// TIA Portal V16 export
// export: Created 2021-11-12T13:33:07.5254994Z, ExportSetting WithDefaults, DisplayName Totally Integrated Automation Portal, DisplayVersion V16 Update 3, DisplayName TIA Portal Version Control Interface, DisplayVersion V16 Update 2, DisplayName TIA Portal Openness, DisplayVersion V16 Update 3, DisplayName SINAMICS Startdrive Advanced, DisplayVersion V16 Update 5, DisplayName SINAMICS Startdrive G130, G150, S120, S150, SINAMICS MV, S210, DisplayVersion V16 Update 5, DisplayName SINAMICS Startdrive G110M, G120, G120C, G120D, G120P, G115D, DisplayVersion V16 Update 5, DisplayName STEP 7 Professional, DisplayVersion V16 Update 3, DisplayName STEP 7 Safety, DisplayVersion V16, DisplayName WinCC UA Professional, DisplayVersion V16 Update 3
DATA_BLOCK "HMI_PARAM_410"   // DB107
{ S7_Optimized_Access := 'TRUE' }
VERSION : 0.1
// stored: AutoNumber true, DBAccessibleFromOPCUA true, IsOnlyStoredInLoadMemory false, IsRetainMemResEnabled false, IsWriteProtectedInAS false, MemoryReserve 100
   VAR
      xxxxx___BinarySensors___xxxxx_1 : Byte;
      "EQ01-BL01" : "UDT_CH_DI_Parameter";   // Sensor for min surface (LSL1440) / Hladina min (LSL1440)
      "EQ01-BL02" : "UDT_CH_DI_Parameter";   // Sensor for max surface (LSH 1441) / Hladina max (LSH 1441)
      "EQ01-MA02_20" : "UDT_CH_DI_Parameter";   // Valve (A1417) - closed
      "EQ01-MA02_24" : "UDT_CH_DI_Parameter";   // Valve (A1417) - opened
      "EQ01-MA03_20" : "UDT_CH_DI_Parameter";   // Valve (A1414) - closed
      "EQ01-MA03_24" : "UDT_CH_DI_Parameter";   // Valve (A1414) - opened
      "EQ01-MA04_20" : "UDT_CH_DI_Parameter";   // Valve (A1411) - closed
      "EQ01-MA04_24" : "UDT_CH_DI_Parameter";   // Valve (A1411) - opened
      xxxxx___BinaryOthers___xxxxx_1 : Byte;
      "UC10-FC21_14" : "UDT_CH_DI_Parameter";   // 230V Hardening tube / 230V Zachlazovací nádrž
      "UC11-FC01_14" : "UDT_CH_DI_Parameter";   // 400V Pump of circulation P31 OK / 400V Čerpadlo cirkulace P31 OK
      xxxxx___AnalogueSensors___xxxxx_1 : Byte;
   END_VAR
   VAR RETAIN
      "EQ01-BT01" : "UDT_CH_AI_Parameter";   // Temperature measurment (TIC 1424) / Měření teploty (TIC 1424)
      "EQ01-BP01" : "UDT_CH_AI_Parameter";   // Tenzometric sond for measure surface (LIC 1430) / Tenzometrická sonda pro měření hladiny (LIC 1430)
      "EQ01-MA03_81" : "UDT_CH_AI_Parameter";   // Meření ventilu A 1414 Zavřeno - otevřeno
   END_VAR
   VAR
      xxxxx___Drives___xxxxx_1 : Byte;
      "EQ01-MA01" : "UDT_Drive1_Parameter";   // Pump of circulation (P31) / Čerpadlo cirkulace (P31)
      "EQ01-MA02" : "UDT_Valve2WB_Parameter";   // Valve with servomotor (A1417) - vypouštění / Ventil se servopohonem (A1417) - vypouštění
      "EQ01-MA03" : "UDT_Valve2WB_Parameter";   // Valve with servomotor (A1414) - chlazení / Ventil se servopohonem (A1414) - chlazení
      "EQ01-MA04" : "UDT_Valve2WB_Parameter";   // Valve with servomotor (A1411) - napouštění / Ventil se servopohonem (A1411) - napouštění
   END_VAR
   VAR RETAIN
      "UC11-TA01" : "UDT_SINAMICS_G120_Parameter";   // Frequence changer ( pro P33) / Frekvenční měnič ( pro P33)
   END_VAR
   VAR
      xxxxx___Alarms___xxxxx : Byte;
      ES : "UDT_DI_Mon_Parameter";   // E-stop
      KF31 : "UDT_DI_Mon_Parameter";   // module KF31
      Alarm_1 { S7_SetPoint := 'True'} : "UDT_DI_Mon_Parameter";   // Sensor Max level active and sensor Min level
      Alarm_2 { S7_SetPoint := 'True'} : "UDT_DI_Mon_Parameter";   // Sensor Min level active and analog level sensor under 10%
      Alarm_3 { S7_SetPoint := 'True'} : "UDT_DI_Mon_Parameter";   // Analog level sensor over 40% and sensor min level not active
      Alarm_4 { S7_SetPoint := 'True'} : "UDT_DI_Mon_Parameter";   // Water temperature high
      Alarm_5 { S7_SetPoint := 'True'} : "UDT_DI_Mon_Parameter";   // Water temperature low
      Alarm_6 { S7_SetPoint := 'True'} : "UDT_DI_Mon_Parameter";   // Water level high
      Alarm_7 { S7_SetPoint := 'True'} : "UDT_DI_Mon_Parameter";   // BSN3 tacts and water level NOK
      Alarm_8 { S7_SetPoint := 'True'} : "UDT_DI_Mon_Parameter";   // Filling and no water level change
      Alarm_9 { S7_SetPoint := 'True'} : "UDT_DI_Mon_Parameter";   // Drain and no water level change
      xxxxx___Others___xxxxx { S7_SetPoint := 'True'} : Byte;
      "EQ01-MA03_RegPar" : Struct   // Cooling regulation
         PGain : Real := 1.0;
         Bias : Real := 50.0;
      END_STRUCT;
   END_VAR
BEGIN
   "EQ01-BT01".RMax := 100.0;
   "EQ01-BT01".RMin := 0.0;
   "EQ01-BP01".RawMax := 4540;
   "EQ01-BP01".RMax := 100.0;
   "EQ01-BP01".RMin := 0.0;
   "EQ01-MA03_81".RMax := 100.0;
   "EQ01-MA03_81".RMin := 0.0;
   "UC11-TA01".RefSpdP2000 := 3000.0;
   "UC11-TA01".RefCurrP2002 := 16.5;
   "UC11-TA01".RefTrqP2003 := 35.85;
END_DATA_BLOCK
